// TIA Portal V17 export
// export: Created 2025-06-26T07:49:41.2483484Z, ExportSetting WithDefaults, DisplayName Totally Integrated Automation Portal, DisplayVersion V17 Update 8, DisplayName TIA Portal Openness, DisplayVersion V17 Update 8, DisplayName TIA Portal Version Control Interface, DisplayVersion V17, DisplayName STEP 7 Professional, DisplayVersion V17 Update 8, DisplayName STEP 7 Safety, DisplayVersion V17 Update 6, DisplayName WinCC Advanced, DisplayVersion V17 Update 8
FUNCTION "State3_PrepareStart" : Void   // FC36, FBD
{ S7_Optimized_Access := 'TRUE' }
VERSION : 0.1
// stored: AutoNumber true, IsIECCheckEnabled false, SetENOAutomatically false, UDAEnableTagReadback false
   VAR_INPUT
      Active : Bool;
   END_VAR
   VAR_OUTPUT
      NextState : Bool;
      Stop : Bool;
      Standby : Bool;
   END_VAR
   VAR_TEMP
      NextStateConditions : Bool;
      PauseHere : Bool;
   END_VAR
   VAR_TEMP   // added for the SCL form of the ladder/FBD networks
      _w1 : Bool;
   END_VAR
BEGIN

REGION Network 1: State number
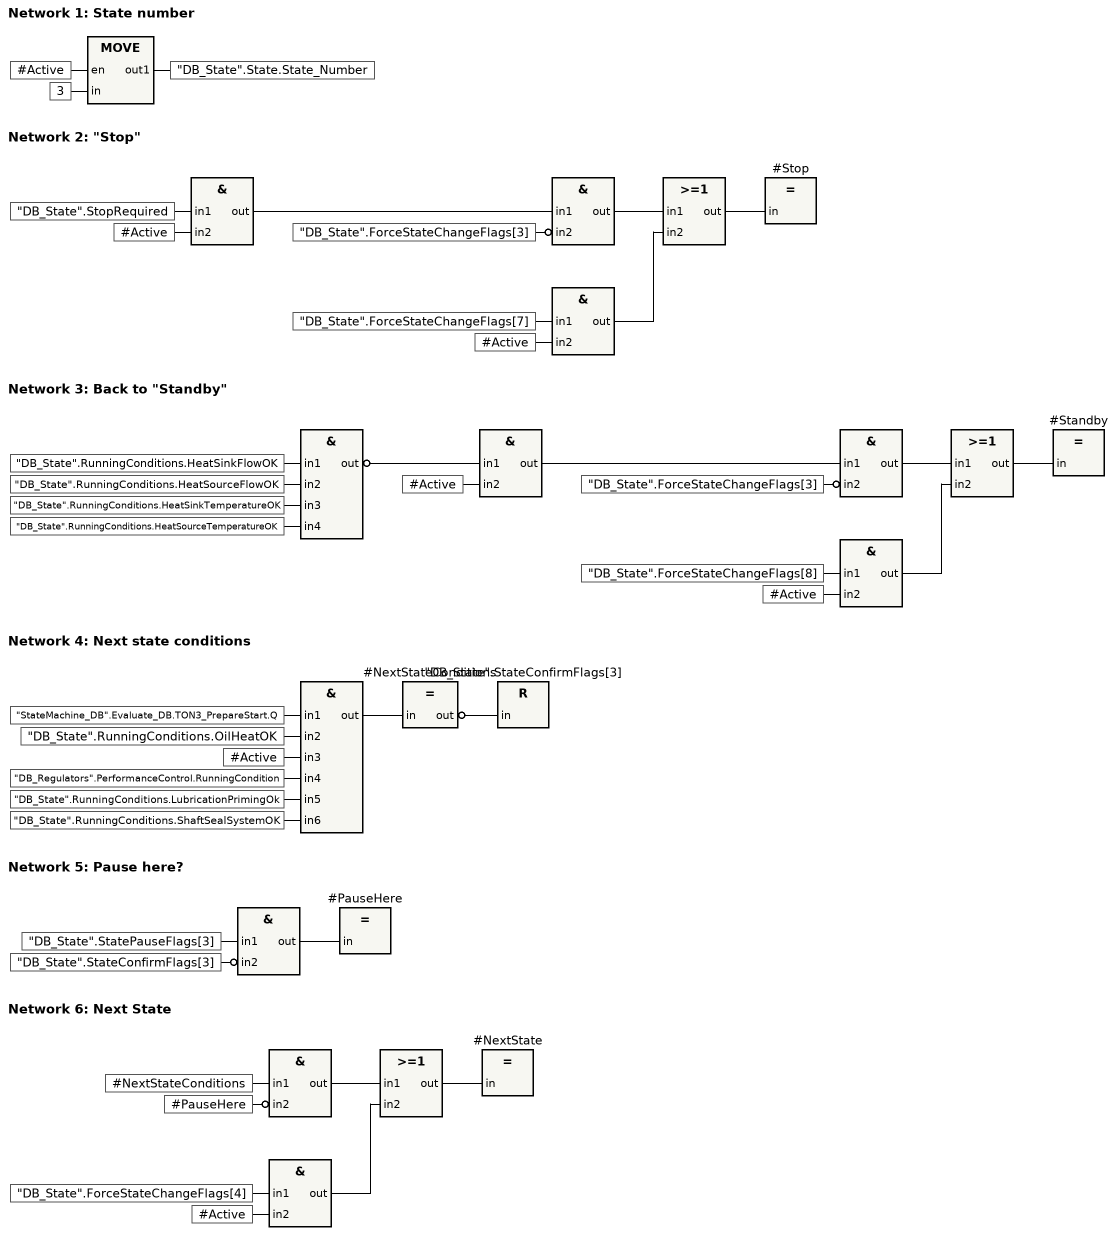
   IF #Active THEN "DB_State".State.State_Number := 3; END_IF;
END_REGION

REGION Network 2: "Stop"
   #Stop := ("DB_State".StopRequired AND #Active AND NOT "DB_State".ForceStateChangeFlags[3]) OR ("DB_State".ForceStateChangeFlags[7] AND #Active);
END_REGION

REGION Network 3: Back to "Standby"
   #Standby := (NOT ("DB_State".RunningConditions.HeatSinkFlowOK AND "DB_State".RunningConditions.HeatSourceFlowOK AND "DB_State".RunningConditions.HeatSinkTemperatureOK AND "DB_State".RunningConditions.HeatSourceTemperatureOK) AND #Active AND NOT "DB_State".ForceStateChangeFlags[3]) OR ("DB_State".ForceStateChangeFlags[8] AND #Active);
END_REGION

REGION Network 4: Next state conditions
   #_w1 := "StateMachine_DB".Evaluate_DB.TON3_PrepareStart.Q AND "DB_State".RunningConditions.OilHeatOK AND #Active AND "DB_Regulators".PerformanceControl.RunningCondition AND "DB_State".RunningConditions.LubricationPrimingOk AND "DB_State".RunningConditions.ShaftSealSystemOK;
   #NextStateConditions := #_w1;
   IF NOT #_w1 THEN "DB_State".StateConfirmFlags[3] := FALSE; END_IF;
END_REGION

REGION Network 5: Pause here?
   // Pause   Confirm  PauseHere
   // 0            0              0
   // 0            1              0
   // 1            0              1
   // 1            1              0
   #PauseHere := "DB_State".StatePauseFlags[3] AND NOT "DB_State".StateConfirmFlags[3];
END_REGION

REGION Network 6: Next State
   #NextState := (#NextStateConditions AND NOT #PauseHere) OR ("DB_State".ForceStateChangeFlags[4] AND #Active);
END_REGION
END_FUNCTION
